FUNCTION F_Add : INT
VAR_INPUT
	a : INT;
	b : INT;
END_VAR

F_Add := a + b;

END_FUNCTION

(* stored: Version 1.1.0.1, ProductVersion 3.1.4026.18
   POU F_Add: Id {00000000-0000-0000-0000-000000000050}, SpecialFunc None *)
